{attribute 'qualified_only'}
VAR_GLOBAL
	StateManager : StateManager;
	iJogFwdButton  : BOOL;	
	iJogRevButton  : BOOL;	
	oJogButtonLight AT %Q* : BOOL;
	oSafetyReset AT %Q* : BOOL;
		iEStopOK AT %I* : BOOL;
END_VAR

(* stored: Version 1.1.0.1, ProductVersion 3.1.4022.11
   GVL Cell: Id {2a2bb7cf-df64-47af-9771-33b156960614} *)
